TYPE PB_Dateneintrag :
STRUCT
	CANAdress 	: BYTE;
	Parameter 	: UINT;	
	Value		: UINT;
	Status		: WORD;
END_STRUCT
END_TYPE

(* stored: Version 1.1.0.1, ProductVersion 3.1.4024.9
   DUT PB_Dateneintrag: Id {9fae1f72-ec7d-4736-a5dd-af095f58c1e6} *)
